FUNCTION_BLOCK FB_AxisDistanceTrigger
VAR_INPUT
	/// reset FB
	bReset				: BOOL;
	/// actual position
	fActualPos			: LREAL;
	/// trigger distance
	fTriggerDistance	: LREAL;
END_VAR
VAR_OUTPUT
	/// trigger output
	Q	: BOOL;
END_VAR
VAR PERSISTENT
	/// distance
	fDistance		: LREAL;
	/// actual ABS position
	fActualAbsPos	: LREAL;
	/// mirror ABS position
	fMirrorAbsPos	: LREAL;
	bInit			: BOOL;
END_VAR

fActualAbsPos := ABS(fActualPos);

IF bReset OR NOT bInit THEN
	bInit := TRUE;
	Q := FALSE;
	fMirrorAbsPos := fActualAbsPos;
	IF bReset THEN	
		fDistance := 0;
	END_IF

END_IF

IF fTriggerDistance <= 0 THEN
	Q := FALSE;
	RETURN;
END_IF

IF ABS(fActualAbsPos - fMirrorAbsPos) > fEpsilon THEN
	fDistance := fDistance + ABS(fActualAbsPos - fMirrorAbsPos);
	fMirrorAbsPos := fActualAbsPos;
END_IF

Q := fDistance >= fTriggerDistance;

END_FUNCTION_BLOCK

(* stored: Version 1.1.0.1, ProductVersion 3.1.4020.12
   POU FB_AxisDistanceTrigger: Id {d3e1280f-14b1-43da-9a9e-aeaa9341d48f}, SpecialFunc None *)
